{attribute 'qualified_only'}
VAR_GLOBAL
	uiStateCmd:UINT;
END_VAR

(* stored: Version 1.1.0.1, ProductVersion 3.1.4022.18
   GVL GVL_CONVERTER: Id {1be9b1cc-51a3-4e1f-9a83-ec22cd679cf3} *)
